// TIA Portal V17 export
// export: Created 2023-12-22T15:08:00.2760816Z, ExportSetting WithDefaults, DisplayName Totally Integrated Automation Portal, DisplayVersion V17, DisplayName TIA Portal Openness, DisplayVersion V17, DisplayName TIA Portal Version Control Interface, DisplayVersion V17, DisplayName STEP 7 Professional, DisplayVersion V17, DisplayName STEP 7 Safety, DisplayVersion V17, DisplayName WinCC Advanced, DisplayVersion V17
FUNCTION_BLOCK "PE_Diag"   // FB4, LAD
{ S7_Optimized_Access := 'FALSE' }
VERSION : 0.1
// stored: AutoNumber true, IsIECCheckEnabled false, SetENOAutomatically false, UDAEnableTagReadback false
   VAR_INPUT
      PE_1 : Real;
      PE_2 : Real;
   END_VAR
   VAR_OUTPUT
      PE : Real;
   END_VAR
   VAR DB_SPECIFIC
      Select : Bool;
      Delta : Real;
      Delta_In : Real;
      Delta_Max { S7_SetPoint := 'True'} : Real := 0.05;
      Warning : Word;
   END_VAR
   VAR_TEMP   // added for the SCL form of the ladder/FBD networks
      _w1 : Bool;
      _w2 : Bool;
   END_VAR
BEGIN

REGION Network 1: Определение расхождения между датчиками
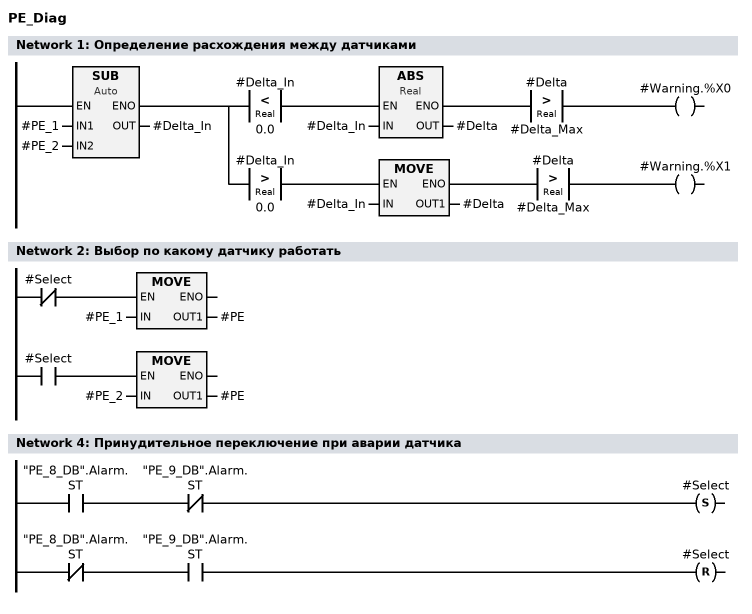
   RUNG wire#powerrail
      Sub(in1 := #PE_1, in2 := #PE_2, out => #Delta_In)
      wire#w1
      { S7_Templates := "SrcType := Real" } LT_Contact(in1 := #Delta_In, in2 := 0.0)
      { S7_Templates := "SrcType := Real" } Abs(in := #Delta_In, out => #Delta)
      { S7_Templates := "SrcType := Real" } GT_Contact(in1 := #Delta, in2 := #Delta_Max)
      Coil( #Warning.%X0 )
   END_RUNG
   RUNG wire#w1
      { S7_Templates := "SrcType := Real" } GT_Contact(in1 := #Delta_In, in2 := 0.0)
      Move(in := #Delta_In, out1 => #Delta)
      { S7_Templates := "SrcType := Real" } GT_Contact(in1 := #Delta, in2 := #Delta_Max)
      Coil( #Warning.%X1 )
   END_RUNG
   // the same network as SCL:
   #Delta_In := #PE_1 - #PE_2;
   #_w1 := #Delta_In < 0.0;
   IF #_w1 THEN #Delta := ABS(#Delta_In); END_IF;
   #Warning.%X0 := #_w1 AND (#Delta > #Delta_Max);
   #_w2 := #Delta_In > 0.0;
   IF #_w2 THEN #Delta := #Delta_In; END_IF;
   #Warning.%X1 := #_w2 AND (#Delta > #Delta_Max);
END_REGION

REGION Network 2: Выбор по какому датчику работать
   RUNG wire#powerrail
      I_Contact( #Select )
      Move(in := #PE_1, out1 => #PE)
   END_RUNG
   RUNG wire#powerrail
      Contact( #Select )
      Move(in := #PE_2, out1 => #PE)
   END_RUNG
   // the same network as SCL:
   IF NOT #Select THEN #PE := #PE_1; END_IF;
   IF #Select THEN #PE := #PE_2; END_IF;
END_REGION

REGION Network 3: Сообщение о расхождении уровней
END_REGION

REGION Network 4: Принудительное переключение при аварии датчика
   RUNG wire#powerrail
      Contact( "PE_8_DB".Alarm.ST )
      I_Contact( "PE_9_DB".Alarm.ST )
      S_Coil( #Select )
   END_RUNG
   RUNG wire#powerrail
      I_Contact( "PE_8_DB".Alarm.ST )
      Contact( "PE_9_DB".Alarm.ST )
      R_Coil( #Select )
   END_RUNG
   // the same network as SCL:
   IF "PE_8_DB".Alarm.ST AND NOT "PE_9_DB".Alarm.ST THEN #Select := TRUE; END_IF;
   IF NOT "PE_8_DB".Alarm.ST AND "PE_9_DB".Alarm.ST THEN #Select := FALSE; END_IF;
END_REGION
END_FUNCTION_BLOCK
